(* PLC project TwinForgePowerFlex525Application, TwinForge TwinForge 0.1.0 *)
(* stored: creationDateTime 2026-07-30T05:53:31.111529+00:00 *)

PROGRAM PLC_PRG
  VAR
    fbPowerFlex525_PF525_01 : TF_PowerFlex525_Core;
    PF525_01_diInp_Source : DINT;
    PF525_01_xInp_PRunFwd : BOOL;
    PF525_01_xInp_PRunRev : BOOL;
    PF525_01_xInp_PJogFwd : BOOL;
    PF525_01_xInp_PJogRev : BOOL;
    PF525_01_xInp_PStop : BOOL;
    PF525_01_xInp_PReset : BOOL;
    PF525_01_rInp_PSpeed : REAL;
    PF525_01_xInp_ORunFwd : BOOL;
    PF525_01_xInp_ORunRev : BOOL;
    PF525_01_xInp_OJogFwd : BOOL;
    PF525_01_xInp_OJogRev : BOOL;
    PF525_01_xInp_OStop : BOOL;
    PF525_01_xInp_OReset : BOOL;
    PF525_01_rInp_OSpeed : REAL;
    PF525_01_xInp_XRunFwd : BOOL;
    PF525_01_xInp_XRunRev : BOOL;
    PF525_01_xInp_XJogFwd : BOOL;
    PF525_01_xInp_XJogRev : BOOL;
    PF525_01_xInp_XStop : BOOL;
    PF525_01_xInp_XReset : BOOL;
    PF525_01_rInp_XSpeed : REAL;
    PF525_01_xInp_MRunFwd : BOOL;
    PF525_01_xInp_MRunRev : BOOL;
    PF525_01_xInp_MJogFwd : BOOL;
    PF525_01_xInp_MJogRev : BOOL;
    PF525_01_xInp_MStop : BOOL;
    PF525_01_xInp_MReset : BOOL;
    PF525_01_rInp_MSpeed : REAL;
    PF525_01_diInp_OvCmd : DINT;
    PF525_01_rInp_OvSpeed : REAL;
    PF525_01_xInp_PSetOverride : BOOL;
    PF525_01_rInp_MPSet : REAL;
    PF525_01_xInp_PermOK : BOOL;
    PF525_01_xInp_NBPermOK : BOOL;
    PF525_01_xInp_IntlkOK : BOOL;
    PF525_01_xInp_NBIntlkOK : BOOL;
    PF525_01_xInp_Bypass : BOOL;
    PF525_01_xInp_RunFwdAvail : BOOL;
    PF525_01_xInp_RunRevAvail : BOOL;
    PF525_01_xInp_JogFwdAvail : BOOL;
    PF525_01_xInp_JogRevAvail : BOOL;
    PF525_01_xInp_Ready : BOOL;
    PF525_01_xInp_Active : BOOL;
    PF525_01_xInp_ENetLogicCtrl : BOOL;
    PF525_01_xInp_KeypadCtrlSts : BOOL;
    PF525_01_xInp_KeypadCtrlCmd : BOOL;
    PF525_01_rInp_MaxSpeed : REAL;
    PF525_01_rInp_JogSpeed : REAL;
    PF525_01_diInp_StartDelayMs : DINT;
    PF525_01_diInp_ElapsedMs : DINT;
    PF525_01_uiOut_LogicCommand : UINT;
    PF525_01_iOut_SpeedCommand : INT;
    PF525_01_rOut_RefSpeed : REAL;
    PF525_01_xOut_PermOK : BOOL;
    PF525_01_xOut_IntlkOK : BOOL;
    PF525_01_xOut_RunFwd : BOOL;
    PF525_01_xOut_RunRev : BOOL;
    PF525_01_xOut_JogFwd : BOOL;
    PF525_01_xOut_JogRev : BOOL;
    PF525_01_xOut_Starting : BOOL;
    PF525_01_xOut_Stopping : BOOL;
    PF525_01_fbModuleBinding : TF_Codesys_ENIP_ModuleBinding;
    PF525_01_xInp_Connected : BOOL;
    PF525_01_xInp_Enabled : BOOL;
    PF525_01_xInp_Faulted : BOOL;
    PF525_01_xInp_DiagnosticAvailable : BOOL;
    PF525_01_xInp_CanReconfigure : BOOL;
    PF525_01_xInp_ReconfigureBusy : BOOL;
    PF525_01_xInp_ReconfigureDone : BOOL;
    PF525_01_xInp_ReconfigureFailed : BOOL;
    PF525_01_xInp_Inhibit : BOOL;
    PF525_01_xInp_Uninhibit : BOOL;
    PF525_01_xOut_Connected : BOOL;
    PF525_01_xOut_Enabled : BOOL;
    PF525_01_xOut_Faulted : BOOL;
    PF525_01_xOut_DiagnosticAvailable : BOOL;
    PF525_01_xOut_RequestReconfigure : BOOL;
    PF525_01_xOut_RequestedEnable : BOOL;
    PF525_01_xOut_ReconfigureBlocked : BOOL;
    PF525_01_xOut_ReconfigureBusy : BOOL;
    PF525_01_xOut_ReconfigureDone : BOOL;
    PF525_01_xOut_ReconfigureFailed : BOOL;
    fbPowerFlex525_PF525_02 : TF_PowerFlex525_Core;
    PF525_02_diInp_Source : DINT;
    PF525_02_xInp_PRunFwd : BOOL;
    PF525_02_xInp_PRunRev : BOOL;
    PF525_02_xInp_PJogFwd : BOOL;
    PF525_02_xInp_PJogRev : BOOL;
    PF525_02_xInp_PStop : BOOL;
    PF525_02_xInp_PReset : BOOL;
    PF525_02_rInp_PSpeed : REAL;
    PF525_02_xInp_ORunFwd : BOOL;
    PF525_02_xInp_ORunRev : BOOL;
    PF525_02_xInp_OJogFwd : BOOL;
    PF525_02_xInp_OJogRev : BOOL;
    PF525_02_xInp_OStop : BOOL;
    PF525_02_xInp_OReset : BOOL;
    PF525_02_rInp_OSpeed : REAL;
    PF525_02_xInp_XRunFwd : BOOL;
    PF525_02_xInp_XRunRev : BOOL;
    PF525_02_xInp_XJogFwd : BOOL;
    PF525_02_xInp_XJogRev : BOOL;
    PF525_02_xInp_XStop : BOOL;
    PF525_02_xInp_XReset : BOOL;
    PF525_02_rInp_XSpeed : REAL;
    PF525_02_xInp_MRunFwd : BOOL;
    PF525_02_xInp_MRunRev : BOOL;
    PF525_02_xInp_MJogFwd : BOOL;
    PF525_02_xInp_MJogRev : BOOL;
    PF525_02_xInp_MStop : BOOL;
    PF525_02_xInp_MReset : BOOL;
    PF525_02_rInp_MSpeed : REAL;
    PF525_02_diInp_OvCmd : DINT;
    PF525_02_rInp_OvSpeed : REAL;
    PF525_02_xInp_PSetOverride : BOOL;
    PF525_02_rInp_MPSet : REAL;
    PF525_02_xInp_PermOK : BOOL;
    PF525_02_xInp_NBPermOK : BOOL;
    PF525_02_xInp_IntlkOK : BOOL;
    PF525_02_xInp_NBIntlkOK : BOOL;
    PF525_02_xInp_Bypass : BOOL;
    PF525_02_xInp_RunFwdAvail : BOOL;
    PF525_02_xInp_RunRevAvail : BOOL;
    PF525_02_xInp_JogFwdAvail : BOOL;
    PF525_02_xInp_JogRevAvail : BOOL;
    PF525_02_xInp_Ready : BOOL;
    PF525_02_xInp_Active : BOOL;
    PF525_02_xInp_ENetLogicCtrl : BOOL;
    PF525_02_xInp_KeypadCtrlSts : BOOL;
    PF525_02_xInp_KeypadCtrlCmd : BOOL;
    PF525_02_rInp_MaxSpeed : REAL;
    PF525_02_rInp_JogSpeed : REAL;
    PF525_02_diInp_StartDelayMs : DINT;
    PF525_02_diInp_ElapsedMs : DINT;
    PF525_02_uiOut_LogicCommand : UINT;
    PF525_02_iOut_SpeedCommand : INT;
    PF525_02_rOut_RefSpeed : REAL;
    PF525_02_xOut_PermOK : BOOL;
    PF525_02_xOut_IntlkOK : BOOL;
    PF525_02_xOut_RunFwd : BOOL;
    PF525_02_xOut_RunRev : BOOL;
    PF525_02_xOut_JogFwd : BOOL;
    PF525_02_xOut_JogRev : BOOL;
    PF525_02_xOut_Starting : BOOL;
    PF525_02_xOut_Stopping : BOOL;
    PF525_02_fbModuleBinding : TF_Codesys_ENIP_ModuleBinding;
    PF525_02_xInp_Connected : BOOL;
    PF525_02_xInp_Enabled : BOOL;
    PF525_02_xInp_Faulted : BOOL;
    PF525_02_xInp_DiagnosticAvailable : BOOL;
    PF525_02_xInp_CanReconfigure : BOOL;
    PF525_02_xInp_ReconfigureBusy : BOOL;
    PF525_02_xInp_ReconfigureDone : BOOL;
    PF525_02_xInp_ReconfigureFailed : BOOL;
    PF525_02_xInp_Inhibit : BOOL;
    PF525_02_xInp_Uninhibit : BOOL;
    PF525_02_xOut_Connected : BOOL;
    PF525_02_xOut_Enabled : BOOL;
    PF525_02_xOut_Faulted : BOOL;
    PF525_02_xOut_DiagnosticAvailable : BOOL;
    PF525_02_xOut_RequestReconfigure : BOOL;
    PF525_02_xOut_RequestedEnable : BOOL;
    PF525_02_xOut_ReconfigureBlocked : BOOL;
    PF525_02_xOut_ReconfigureBusy : BOOL;
    PF525_02_xOut_ReconfigureDone : BOOL;
    PF525_02_xOut_ReconfigureFailed : BOOL;
    PF525_01_fbReconfigure : DED.Reconfigure;
    PF525_01_xObservedEnabled : BOOL;
    PF525_01_xObservedDiagnosticAvailable : BOOL;
    PF525_01_sObservedDiagnostic : STRING(255);
    PF525_01_eObservedDeviceState : DED.DEVICE_STATE;
    PF525_01_eObservedReconfigureError : DED.ERROR;
    PF525_02_fbReconfigure : DED.Reconfigure;
    PF525_02_xObservedEnabled : BOOL;
    PF525_02_xObservedDiagnosticAvailable : BOOL;
    PF525_02_sObservedDiagnostic : STRING(255);
    PF525_02_eObservedDeviceState : DED.DEVICE_STATE;
    PF525_02_eObservedReconfigureError : DED.ERROR;
  END_VAR

                  PF525_01_xObservedEnabled := Dev_PF525_01.Enable;
PF525_01_xObservedDiagnosticAvailable := Dev_PF525_01.xDiagnosticAvailable;
PF525_01_sObservedDiagnostic := Dev_PF525_01.sDiagString;
PF525_01_eObservedDeviceState := Dev_PF525_01.GetDeviceState();

PF525_01_xInp_CanReconfigure := DED.CanReconfigure(
    itfNode := Dev_PF525_01
);

PF525_01_xInp_Connected :=
    (Dev_PF525_01.eState = IoDrvEtherNetIP.AdapterState.RUNNING)
    AND
    (PF525_01_eObservedDeviceState = DED.DEVICE_STATE.RUNNING);
PF525_01_xInp_Enabled := Dev_PF525_01.Enable;
PF525_01_xInp_Faulted :=
    (Dev_PF525_01.eState = IoDrvEtherNetIP.AdapterState.BUS_ERROR)
    OR
    (Dev_PF525_01.eState = IoDrvEtherNetIP.AdapterState.ERROR)
    OR
    (PF525_01_eObservedDeviceState = DED.DEVICE_STATE.ERROR);
PF525_01_xInp_DiagnosticAvailable := Dev_PF525_01.xDiagnosticAvailable;
PF525_01_xInp_ReconfigureBusy := PF525_01_fbReconfigure.xBusy;
PF525_01_xInp_ReconfigureDone := PF525_01_fbReconfigure.xDone;
PF525_01_xInp_ReconfigureFailed := PF525_01_fbReconfigure.xError;
PF525_01_eObservedReconfigureError := PF525_01_fbReconfigure.eError;

fbPowerFlex525_PF525_01(
    Inp_Source := PF525_01_diInp_Source,
    Inp_PRunFwd := PF525_01_xInp_PRunFwd,
    Inp_PRunRev := PF525_01_xInp_PRunRev,
    Inp_PJogFwd := PF525_01_xInp_PJogFwd,
    Inp_PJogRev := PF525_01_xInp_PJogRev,
    Inp_PStop := PF525_01_xInp_PStop,
    Inp_PReset := PF525_01_xInp_PReset,
    Inp_PSpeed := PF525_01_rInp_PSpeed,
    Inp_ORunFwd := PF525_01_xInp_ORunFwd,
    Inp_ORunRev := PF525_01_xInp_ORunRev,
    Inp_OJogFwd := PF525_01_xInp_OJogFwd,
    Inp_OJogRev := PF525_01_xInp_OJogRev,
    Inp_OStop := PF525_01_xInp_OStop,
    Inp_OReset := PF525_01_xInp_OReset,
    Inp_OSpeed := PF525_01_rInp_OSpeed,
    Inp_XRunFwd := PF525_01_xInp_XRunFwd,
    Inp_XRunRev := PF525_01_xInp_XRunRev,
    Inp_XJogFwd := PF525_01_xInp_XJogFwd,
    Inp_XJogRev := PF525_01_xInp_XJogRev,
    Inp_XStop := PF525_01_xInp_XStop,
    Inp_XReset := PF525_01_xInp_XReset,
    Inp_XSpeed := PF525_01_rInp_XSpeed,
    Inp_MRunFwd := PF525_01_xInp_MRunFwd,
    Inp_MRunRev := PF525_01_xInp_MRunRev,
    Inp_MJogFwd := PF525_01_xInp_MJogFwd,
    Inp_MJogRev := PF525_01_xInp_MJogRev,
    Inp_MStop := PF525_01_xInp_MStop,
    Inp_MReset := PF525_01_xInp_MReset,
    Inp_MSpeed := PF525_01_rInp_MSpeed,
    Inp_OvCmd := PF525_01_diInp_OvCmd,
    Inp_OvSpeed := PF525_01_rInp_OvSpeed,
    Inp_PSetOverride := PF525_01_xInp_PSetOverride,
    Inp_MPSet := PF525_01_rInp_MPSet,
    Inp_PermOK := PF525_01_xInp_PermOK,
    Inp_NBPermOK := PF525_01_xInp_NBPermOK,
    Inp_IntlkOK := PF525_01_xInp_IntlkOK,
    Inp_NBIntlkOK := PF525_01_xInp_NBIntlkOK,
    Inp_Bypass := PF525_01_xInp_Bypass,
    Inp_RunFwdAvail := PF525_01_xInp_RunFwdAvail,
    Inp_RunRevAvail := PF525_01_xInp_RunRevAvail,
    Inp_JogFwdAvail := PF525_01_xInp_JogFwdAvail,
    Inp_JogRevAvail := PF525_01_xInp_JogRevAvail,
    Inp_Ready := PF525_01_xInp_Ready,
    Inp_Active := PF525_01_xInp_Active,
    Inp_ENetLogicCtrl := PF525_01_xInp_ENetLogicCtrl,
    Inp_KeypadCtrlSts := PF525_01_xInp_KeypadCtrlSts,
    Inp_KeypadCtrlCmd := PF525_01_xInp_KeypadCtrlCmd,
    Inp_MaxSpeed := PF525_01_rInp_MaxSpeed,
    Inp_JogSpeed := PF525_01_rInp_JogSpeed,
    Inp_StartDelayMs := PF525_01_diInp_StartDelayMs,
    Inp_ElapsedMs := PF525_01_diInp_ElapsedMs,
    Out_LogicCommand => PF525_01_uiOut_LogicCommand,
    Out_SpeedCommand => PF525_01_iOut_SpeedCommand,
    Out_RefSpeed => PF525_01_rOut_RefSpeed,
    Out_PermOK => PF525_01_xOut_PermOK,
    Out_IntlkOK => PF525_01_xOut_IntlkOK,
    Out_RunFwd => PF525_01_xOut_RunFwd,
    Out_RunRev => PF525_01_xOut_RunRev,
    Out_JogFwd => PF525_01_xOut_JogFwd,
    Out_JogRev => PF525_01_xOut_JogRev,
    Out_Starting => PF525_01_xOut_Starting,
    Out_Stopping => PF525_01_xOut_Stopping
);

PF525_01_fbModuleBinding(
    Inp_Connected := PF525_01_xInp_Connected,
    Inp_Enabled := PF525_01_xInp_Enabled,
    Inp_Faulted := PF525_01_xInp_Faulted,
    Inp_DiagnosticAvailable := PF525_01_xInp_DiagnosticAvailable,
    Inp_CanReconfigure := PF525_01_xInp_CanReconfigure,
    Inp_ReconfigureBusy := PF525_01_xInp_ReconfigureBusy,
    Inp_ReconfigureDone := PF525_01_xInp_ReconfigureDone,
    Inp_ReconfigureFailed := PF525_01_xInp_ReconfigureFailed,
    Inp_Inhibit := PF525_01_xInp_Inhibit,
    Inp_Uninhibit := PF525_01_xInp_Uninhibit,
    Out_Connected => PF525_01_xOut_Connected,
    Out_Enabled => PF525_01_xOut_Enabled,
    Out_Faulted => PF525_01_xOut_Faulted,
    Out_DiagnosticAvailable => PF525_01_xOut_DiagnosticAvailable,
    Out_RequestReconfigure => PF525_01_xOut_RequestReconfigure,
    Out_RequestedEnable => PF525_01_xOut_RequestedEnable,
    Out_ReconfigureBlocked => PF525_01_xOut_ReconfigureBlocked,
    Out_ReconfigureBusy => PF525_01_xOut_ReconfigureBusy,
    Out_ReconfigureDone => PF525_01_xOut_ReconfigureDone,
    Out_ReconfigureFailed => PF525_01_xOut_ReconfigureFailed
);

IF PF525_01_xOut_RequestReconfigure THEN
    Dev_PF525_01.Enable := PF525_01_xOut_RequestedEnable;
END_IF;

PF525_01_fbReconfigure(
    xExecute := PF525_01_xOut_RequestReconfigure,
    itfNode := Dev_PF525_01
);

PF525_02_xObservedEnabled := Dev_PF525_02.Enable;
PF525_02_xObservedDiagnosticAvailable := Dev_PF525_02.xDiagnosticAvailable;
PF525_02_sObservedDiagnostic := Dev_PF525_02.sDiagString;
PF525_02_eObservedDeviceState := Dev_PF525_02.GetDeviceState();

PF525_02_xInp_CanReconfigure := DED.CanReconfigure(
    itfNode := Dev_PF525_02
);

PF525_02_xInp_Connected :=
    (Dev_PF525_02.eState = IoDrvEtherNetIP.AdapterState.RUNNING)
    AND
    (PF525_02_eObservedDeviceState = DED.DEVICE_STATE.RUNNING);
PF525_02_xInp_Enabled := Dev_PF525_02.Enable;
PF525_02_xInp_Faulted :=
    (Dev_PF525_02.eState = IoDrvEtherNetIP.AdapterState.BUS_ERROR)
    OR
    (Dev_PF525_02.eState = IoDrvEtherNetIP.AdapterState.ERROR)
    OR
    (PF525_02_eObservedDeviceState = DED.DEVICE_STATE.ERROR);
PF525_02_xInp_DiagnosticAvailable := Dev_PF525_02.xDiagnosticAvailable;
PF525_02_xInp_ReconfigureBusy := PF525_02_fbReconfigure.xBusy;
PF525_02_xInp_ReconfigureDone := PF525_02_fbReconfigure.xDone;
PF525_02_xInp_ReconfigureFailed := PF525_02_fbReconfigure.xError;
PF525_02_eObservedReconfigureError := PF525_02_fbReconfigure.eError;

fbPowerFlex525_PF525_02(
    Inp_Source := PF525_02_diInp_Source,
    Inp_PRunFwd := PF525_02_xInp_PRunFwd,
    Inp_PRunRev := PF525_02_xInp_PRunRev,
    Inp_PJogFwd := PF525_02_xInp_PJogFwd,
    Inp_PJogRev := PF525_02_xInp_PJogRev,
    Inp_PStop := PF525_02_xInp_PStop,
    Inp_PReset := PF525_02_xInp_PReset,
    Inp_PSpeed := PF525_02_rInp_PSpeed,
    Inp_ORunFwd := PF525_02_xInp_ORunFwd,
    Inp_ORunRev := PF525_02_xInp_ORunRev,
    Inp_OJogFwd := PF525_02_xInp_OJogFwd,
    Inp_OJogRev := PF525_02_xInp_OJogRev,
    Inp_OStop := PF525_02_xInp_OStop,
    Inp_OReset := PF525_02_xInp_OReset,
    Inp_OSpeed := PF525_02_rInp_OSpeed,
    Inp_XRunFwd := PF525_02_xInp_XRunFwd,
    Inp_XRunRev := PF525_02_xInp_XRunRev,
    Inp_XJogFwd := PF525_02_xInp_XJogFwd,
    Inp_XJogRev := PF525_02_xInp_XJogRev,
    Inp_XStop := PF525_02_xInp_XStop,
    Inp_XReset := PF525_02_xInp_XReset,
    Inp_XSpeed := PF525_02_rInp_XSpeed,
    Inp_MRunFwd := PF525_02_xInp_MRunFwd,
    Inp_MRunRev := PF525_02_xInp_MRunRev,
    Inp_MJogFwd := PF525_02_xInp_MJogFwd,
    Inp_MJogRev := PF525_02_xInp_MJogRev,
    Inp_MStop := PF525_02_xInp_MStop,
    Inp_MReset := PF525_02_xInp_MReset,
    Inp_MSpeed := PF525_02_rInp_MSpeed,
    Inp_OvCmd := PF525_02_diInp_OvCmd,
    Inp_OvSpeed := PF525_02_rInp_OvSpeed,
    Inp_PSetOverride := PF525_02_xInp_PSetOverride,
    Inp_MPSet := PF525_02_rInp_MPSet,
    Inp_PermOK := PF525_02_xInp_PermOK,
    Inp_NBPermOK := PF525_02_xInp_NBPermOK,
    Inp_IntlkOK := PF525_02_xInp_IntlkOK,
    Inp_NBIntlkOK := PF525_02_xInp_NBIntlkOK,
    Inp_Bypass := PF525_02_xInp_Bypass,
    Inp_RunFwdAvail := PF525_02_xInp_RunFwdAvail,
    Inp_RunRevAvail := PF525_02_xInp_RunRevAvail,
    Inp_JogFwdAvail := PF525_02_xInp_JogFwdAvail,
    Inp_JogRevAvail := PF525_02_xInp_JogRevAvail,
    Inp_Ready := PF525_02_xInp_Ready,
    Inp_Active := PF525_02_xInp_Active,
    Inp_ENetLogicCtrl := PF525_02_xInp_ENetLogicCtrl,
    Inp_KeypadCtrlSts := PF525_02_xInp_KeypadCtrlSts,
    Inp_KeypadCtrlCmd := PF525_02_xInp_KeypadCtrlCmd,
    Inp_MaxSpeed := PF525_02_rInp_MaxSpeed,
    Inp_JogSpeed := PF525_02_rInp_JogSpeed,
    Inp_StartDelayMs := PF525_02_diInp_StartDelayMs,
    Inp_ElapsedMs := PF525_02_diInp_ElapsedMs,
    Out_LogicCommand => PF525_02_uiOut_LogicCommand,
    Out_SpeedCommand => PF525_02_iOut_SpeedCommand,
    Out_RefSpeed => PF525_02_rOut_RefSpeed,
    Out_PermOK => PF525_02_xOut_PermOK,
    Out_IntlkOK => PF525_02_xOut_IntlkOK,
    Out_RunFwd => PF525_02_xOut_RunFwd,
    Out_RunRev => PF525_02_xOut_RunRev,
    Out_JogFwd => PF525_02_xOut_JogFwd,
    Out_JogRev => PF525_02_xOut_JogRev,
    Out_Starting => PF525_02_xOut_Starting,
    Out_Stopping => PF525_02_xOut_Stopping
);

PF525_02_fbModuleBinding(
    Inp_Connected := PF525_02_xInp_Connected,
    Inp_Enabled := PF525_02_xInp_Enabled,
    Inp_Faulted := PF525_02_xInp_Faulted,
    Inp_DiagnosticAvailable := PF525_02_xInp_DiagnosticAvailable,
    Inp_CanReconfigure := PF525_02_xInp_CanReconfigure,
    Inp_ReconfigureBusy := PF525_02_xInp_ReconfigureBusy,
    Inp_ReconfigureDone := PF525_02_xInp_ReconfigureDone,
    Inp_ReconfigureFailed := PF525_02_xInp_ReconfigureFailed,
    Inp_Inhibit := PF525_02_xInp_Inhibit,
    Inp_Uninhibit := PF525_02_xInp_Uninhibit,
    Out_Connected => PF525_02_xOut_Connected,
    Out_Enabled => PF525_02_xOut_Enabled,
    Out_Faulted => PF525_02_xOut_Faulted,
    Out_DiagnosticAvailable => PF525_02_xOut_DiagnosticAvailable,
    Out_RequestReconfigure => PF525_02_xOut_RequestReconfigure,
    Out_RequestedEnable => PF525_02_xOut_RequestedEnable,
    Out_ReconfigureBlocked => PF525_02_xOut_ReconfigureBlocked,
    Out_ReconfigureBusy => PF525_02_xOut_ReconfigureBusy,
    Out_ReconfigureDone => PF525_02_xOut_ReconfigureDone,
    Out_ReconfigureFailed => PF525_02_xOut_ReconfigureFailed
);

IF PF525_02_xOut_RequestReconfigure THEN
    Dev_PF525_02.Enable := PF525_02_xOut_RequestedEnable;
END_IF;

PF525_02_fbReconfigure(
    xExecute := PF525_02_xOut_RequestReconfigure,
    itfNode := Dev_PF525_02
);
                
END_PROGRAM

FUNCTION_BLOCK TF_PowerFlex525_Core
  VAR_INPUT
    Inp_Source : DINT;
    Inp_PRunFwd : BOOL;
    Inp_PRunRev : BOOL;
    Inp_PJogFwd : BOOL;
    Inp_PJogRev : BOOL;
    Inp_PStop : BOOL;
    Inp_PReset : BOOL;
    Inp_PSpeed : REAL;
    Inp_ORunFwd : BOOL;
    Inp_ORunRev : BOOL;
    Inp_OJogFwd : BOOL;
    Inp_OJogRev : BOOL;
    Inp_OStop : BOOL;
    Inp_OReset : BOOL;
    Inp_OSpeed : REAL;
    Inp_XRunFwd : BOOL;
    Inp_XRunRev : BOOL;
    Inp_XJogFwd : BOOL;
    Inp_XJogRev : BOOL;
    Inp_XStop : BOOL;
    Inp_XReset : BOOL;
    Inp_XSpeed : REAL;
    Inp_MRunFwd : BOOL;
    Inp_MRunRev : BOOL;
    Inp_MJogFwd : BOOL;
    Inp_MJogRev : BOOL;
    Inp_MStop : BOOL;
    Inp_MReset : BOOL;
    Inp_MSpeed : REAL;
    Inp_OvCmd : DINT;
    Inp_OvSpeed : REAL;
    Inp_PSetOverride : BOOL;
    Inp_MPSet : REAL;
    Inp_PermOK : BOOL;
    Inp_NBPermOK : BOOL;
    Inp_IntlkOK : BOOL;
    Inp_NBIntlkOK : BOOL;
    Inp_Bypass : BOOL;
    Inp_RunFwdAvail : BOOL;
    Inp_RunRevAvail : BOOL;
    Inp_JogFwdAvail : BOOL;
    Inp_JogRevAvail : BOOL;
    Inp_Ready : BOOL;
    Inp_Active : BOOL;
    Inp_ENetLogicCtrl : BOOL;
    Inp_KeypadCtrlSts : BOOL;
    Inp_KeypadCtrlCmd : BOOL;
    Inp_MaxSpeed : REAL;
    Inp_JogSpeed : REAL;
    Inp_StartDelayMs : DINT;
    Inp_ElapsedMs : DINT;
  END_VAR
  VAR_OUTPUT
    Out_LogicCommand : UINT;
    Out_SpeedCommand : INT;
    Out_RefSpeed : REAL;
    Out_PermOK : BOOL;
    Out_IntlkOK : BOOL;
    Out_RunFwd : BOOL;
    Out_RunRev : BOOL;
    Out_JogFwd : BOOL;
    Out_JogRev : BOOL;
    Out_Starting : BOOL;
    Out_Stopping : BOOL;
  END_VAR
  VAR
    RunFwd : BOOL;
    RunRev : BOOL;
    StartElapsedMs : DINT;
    TimerDone : BOOL;
    StopCmd : BOOL;
    StartCmd : BOOL;
    JogCmd : BOOL;
    ResetCmd : BOOL;
    SpeedRef : REAL;
  END_VAR

                  Out_PermOK := ((Inp_PermOK OR Inp_Bypass) AND Inp_NBPermOK);
Out_IntlkOK := ((Inp_IntlkOK OR Inp_Bypass) AND Inp_NBIntlkOK);
IF (Inp_Source = 1) THEN
    IF Inp_PSetOverride THEN
        Out_RefSpeed := Inp_MPSet;
    ELSE
        Out_RefSpeed := Inp_PSpeed;
    END_IF;
    RunFwd := (((Inp_PRunFwd AND (Out_PermOK OR RunFwd)) AND Out_IntlkOK) AND NOT (Inp_PStop));
    RunRev := (((Inp_PRunRev AND (Out_PermOK OR RunRev)) AND Out_IntlkOK) AND NOT (Inp_PStop));
ELSIF (Inp_Source = 2) THEN
    Out_RefSpeed := Inp_OSpeed;
    RunFwd := (((RunFwd OR (((Inp_ORunFwd AND Inp_RunFwdAvail) AND Out_PermOK) AND NOT (Inp_ORunRev))) AND Out_IntlkOK) AND NOT (Inp_OStop));
    RunRev := (((RunRev OR (((Inp_ORunRev AND Inp_RunRevAvail) AND Out_PermOK) AND NOT (Inp_ORunFwd))) AND Out_IntlkOK) AND NOT (Inp_OStop));
ELSIF (Inp_Source = 3) THEN
    Out_RefSpeed := Inp_XSpeed;
    RunFwd := (((RunFwd OR (((Inp_XRunFwd AND Inp_RunFwdAvail) AND Out_PermOK) AND NOT (Inp_XRunRev))) AND Out_IntlkOK) AND NOT (Inp_XStop));
    RunRev := (((RunRev OR (((Inp_XRunRev AND Inp_RunRevAvail) AND Out_PermOK) AND NOT (Inp_XRunFwd))) AND Out_IntlkOK) AND NOT (Inp_XStop));
ELSIF (Inp_Source = 4) THEN
    Out_RefSpeed := Inp_OvSpeed;
    IF ((Inp_OvCmd = 1) OR NOT (Out_IntlkOK)) THEN
        RunFwd := FALSE;
        RunRev := FALSE;
    ELSIF ((Inp_OvCmd = 2) AND Out_PermOK) THEN
        RunRev := FALSE;
        RunFwd := TRUE;
    ELSIF ((Inp_OvCmd = 3) AND Out_PermOK) THEN
        RunFwd := FALSE;
        RunRev := TRUE;
    END_IF;
ELSIF (Inp_Source = 5) THEN
    Out_RefSpeed := Inp_MSpeed;
    RunFwd := (((RunFwd OR (((Inp_MRunFwd AND Inp_RunFwdAvail) AND Out_PermOK) AND NOT (Inp_MRunRev))) AND Out_IntlkOK) AND NOT (Inp_MStop));
    RunRev := (((RunRev OR (((Inp_MRunRev AND Inp_RunRevAvail) AND Out_PermOK) AND NOT (Inp_MRunFwd))) AND Out_IntlkOK) AND NOT (Inp_MStop));
ELSE
    Out_RefSpeed := 0.0;
    RunFwd := FALSE;
    RunRev := FALSE;
END_IF;
Out_JogFwd := (((Inp_JogFwdAvail AND Out_PermOK) AND (((((Inp_Source = 2) AND Inp_OJogFwd) AND NOT (Inp_OJogRev)) OR (((Inp_Source = 3) AND Inp_XJogFwd) AND NOT (Inp_XJogRev))) OR (((Inp_Source = 5) AND Inp_MJogFwd) AND NOT (Inp_MJogRev)))) OR (((Inp_Source = 1) AND Inp_PJogFwd) AND NOT (Inp_PJogRev)));
Out_JogRev := (((Inp_JogRevAvail AND Out_PermOK) AND (((((Inp_Source = 2) AND Inp_OJogRev) AND NOT (Inp_OJogFwd)) OR (((Inp_Source = 3) AND Inp_XJogRev) AND NOT (Inp_XJogFwd))) OR (((Inp_Source = 5) AND Inp_MJogRev) AND NOT (Inp_MJogFwd)))) OR (((Inp_Source = 1) AND Inp_PJogRev) AND NOT (Inp_PJogFwd)));
IF (RunFwd OR RunRev) THEN
    StartElapsedMs := (StartElapsedMs + Inp_ElapsedMs);
    IF (StartElapsedMs >= Inp_StartDelayMs) THEN
        StartElapsedMs := Inp_StartDelayMs;
        TimerDone := TRUE;
    ELSE
        TimerDone := FALSE;
    END_IF;
ELSE
    StartElapsedMs := 0;
    TimerDone := FALSE;
END_IF;
Out_Starting := ((RunFwd OR RunRev) AND NOT (TimerDone));
StopCmd := ((Inp_Active AND Inp_ENetLogicCtrl) AND NOT (((((Inp_KeypadCtrlSts OR RunFwd) OR RunRev) OR Out_JogFwd) OR Out_JogRev)));
StartCmd := (((Inp_Ready AND TimerDone) AND NOT (StopCmd)) AND (((RunFwd OR RunRev) OR Out_JogFwd) OR Out_JogRev));
JogCmd := ((Inp_Ready AND NOT (((StopCmd OR RunFwd) OR RunRev))) AND (Out_JogFwd OR Out_JogRev));
ResetCmd := (((Inp_PReset OR Inp_OReset) OR Inp_XReset) OR Inp_MReset);
Out_LogicCommand := 0;
IF StopCmd THEN
    Out_LogicCommand := (Out_LogicCommand + 1);
END_IF;
IF StartCmd THEN
    Out_LogicCommand := (Out_LogicCommand + 2);
END_IF;
IF JogCmd THEN
    Out_LogicCommand := (Out_LogicCommand + 4);
END_IF;
IF ResetCmd THEN
    Out_LogicCommand := (Out_LogicCommand + 8);
END_IF;
IF (RunFwd OR Out_JogFwd) THEN
    Out_LogicCommand := (Out_LogicCommand + 16);
END_IF;
IF (RunRev OR Out_JogRev) THEN
    Out_LogicCommand := (Out_LogicCommand + 32);
END_IF;
IF Inp_KeypadCtrlCmd THEN
    Out_LogicCommand := (Out_LogicCommand + 64);
END_IF;
IF (Out_JogFwd OR Out_JogRev) THEN
    SpeedRef := Inp_JogSpeed;
ELSE
    SpeedRef := Out_RefSpeed;
END_IF;
IF (SpeedRef < 0.0) THEN
    SpeedRef := 0.0;
ELSIF (SpeedRef > Inp_MaxSpeed) THEN
    SpeedRef := Inp_MaxSpeed;
END_IF;
Out_SpeedCommand := REAL_TO_INT((SpeedRef * 100.0));
Out_RunFwd := RunFwd;
Out_RunRev := RunRev;
Out_Stopping := (Inp_Active AND NOT ((((RunFwd OR RunRev) OR Out_JogFwd) OR Out_JogRev)));
                
END_FUNCTION_BLOCK

FUNCTION_BLOCK TF_Codesys_ENIP_ModuleBinding
  VAR_INPUT
    Inp_Connected : BOOL;
    Inp_Enabled : BOOL;
    Inp_Faulted : BOOL;
    Inp_DiagnosticAvailable : BOOL;
    Inp_CanReconfigure : BOOL;
    Inp_ReconfigureBusy : BOOL;
    Inp_ReconfigureDone : BOOL;
    Inp_ReconfigureFailed : BOOL;
    Inp_Inhibit : BOOL;
    Inp_Uninhibit : BOOL;
  END_VAR
  VAR_OUTPUT
    Out_Connected : BOOL;
    Out_Enabled : BOOL;
    Out_Faulted : BOOL;
    Out_DiagnosticAvailable : BOOL;
    Out_RequestReconfigure : BOOL;
    Out_RequestedEnable : BOOL;
    Out_ReconfigureBlocked : BOOL;
    Out_ReconfigureBusy : BOOL;
    Out_ReconfigureDone : BOOL;
    Out_ReconfigureFailed : BOOL;
  END_VAR
  VAR
    CommandLatch : BOOL;
  END_VAR

                  Out_Connected := Inp_Connected;
Out_Enabled := Inp_Enabled;
Out_Faulted := Inp_Faulted;
Out_DiagnosticAvailable := Inp_DiagnosticAvailable;
Out_ReconfigureBusy := Inp_ReconfigureBusy;
Out_ReconfigureDone := Inp_ReconfigureDone;
Out_ReconfigureFailed := Inp_ReconfigureFailed;
Out_RequestReconfigure := FALSE;
IF ((Inp_Inhibit OR Inp_Uninhibit) AND NOT (CommandLatch)) THEN
    IF (Inp_CanReconfigure AND NOT (Inp_ReconfigureBusy)) THEN
        Out_RequestedEnable := NOT (Inp_Inhibit);
        Out_RequestReconfigure := TRUE;
        Out_ReconfigureBlocked := FALSE;
    ELSE
        Out_ReconfigureBlocked := TRUE;
    END_IF;
END_IF;
IF Inp_ReconfigureDone THEN
    Out_ReconfigureBlocked := FALSE;
END_IF;
CommandLatch := (Inp_Inhibit OR Inp_Uninhibit);
                
END_FUNCTION_BLOCK

CONFIGURATION Application
  RESOURCE Application ON PLC
    TASK MainTask(INTERVAL := T#20ms, PRIORITY := 1);
    PROGRAM PLC_PRG WITH MainTask : PLC_PRG;
  END_RESOURCE
END_CONFIGURATION
